// TIA Portal V18 export
TYPE "typeGuideAxisBool"
// stored: IsFailsafeCompliant false
   STRUCT
      M1Z : Bool;
      M2Y : Bool;
      M3X : Bool;
      M4O1 : Bool;
      M5O2 : Bool;
      M6doors : Bool;
   END_STRUCT;
END_TYPE
